// TIA Portal V20 export
TYPE "LER_TypeFATMode_Sampling_ProcessValue"
// stored: Access Published
   STRUCT
      CellCount : Int;
      SelectCount_ProcessValue : Int;
   END_STRUCT;
END_TYPE
